// TIA Portal V17 export
// export: Created 2026-04-13T11:12:44.194684Z, ExportSetting WithDefaults, DisplayName Totally Integrated Automation Portal, DisplayVersion V17 Update 4, DisplayName TIA Portal Openness, DisplayVersion V17 Update 4, DisplayName TIA Portal Version Control Interface, DisplayVersion V17, DisplayName SINAMICS Startdrive Advanced, DisplayVersion V17, DisplayName SINAMICS Startdrive G130, G150, S120, S150, SINAMICS MV, S210, DisplayVersion V17, DisplayName SINAMICS Startdrive G110M, G120, G120C, G120D, G120P, G115D, DisplayVersion V17, DisplayName STEP 7 Professional, DisplayVersion V17 Update 4, DisplayName STEP 7 Safety, DisplayVersion V17, DisplayName WinCC Professional, DisplayVersion V17 Update 4
FUNCTION_BLOCK "15-称重系统"   // FB47, LAD
{ S7_Optimized_Access := 'TRUE' }
VERSION : 0.1
// stored: AutoNumber true, IsIECCheckEnabled false, IsRetainMemResEnabled false, MemoryReserve 100, SetENOAutomatically false, UDAEnableTagReadback false
   VAR_OUTPUT
      管道已堵塞 : Bool;
   END_VAR
   VAR_IN_OUT
      PLUS_1S : Bool;
      YX允许值 : Int;
      超时时间 : Time := T#30S;
      FK反馈值 : Int;
      FK初次反馈值 : Int;
      FK二次反馈值 : Int;
      i : UDInt;
      TTIME : Time;
   END_VAR
   VAR
      t1 : TON_TIME;
      RT1 : R_TRIG;
      RT2 : R_TRIG;
      CZ差值 : Int;
      TT : IEC_TIMER;
   END_VAR
   VAR_TEMP
      TM_FZ : Bool;
      j : Int;
   END_VAR
BEGIN

REGION Network 1 (SCL)
   // 间隔时间，通针开关

   #t1(IN := (#CZ差值> #YX允许值) ,
       PT := #超时时间,
       Q=>#管道已堵塞);
   #TTIME := #t1.ET;

   #RT1(CLK := "Clock_1Hz");

   IF  #RT1.Q THEN
       #i += 1;
   END_IF;

   IF #i >= 60 THEN
       #i := 0;
   END_IF;

   IF #i > 0 AND #i < 30 THEN
       #FK初次反馈值 := #FK反馈值;
   END_IF;

   IF #i < 60 AND #i > 30 THEN
       #FK二次反馈值 := #FK反馈值;
   END_IF;

   #CZ差值 := ABS(#FK初次反馈值 - #FK二次反馈值);
END_REGION
END_FUNCTION_BLOCK
